FUNCTION_BLOCK CiA_DS402Statusword_INOVANCE EXTENDS CiA_DS402Statusword
VAR_INPUT
END_VAR
VAR_OUTPUT	
	TargetReached			: BOOL; // Bit 10 commonly used for in target position, velocity ect.
	HomeFound				: BOOL; // Bit 15: 
END_VAR

METHOD PUBLIC readStatusword : BOOL
VAR_INPUT
	Statusword 		:	UINT;
END_VAR
SUPER^.readStatusword(Statusword);

TargetReached												:= Statusword.10;
HomeFound													:= Statusword.15;
readStatusword												:= TRUE;
END_METHOD

END_FUNCTION_BLOCK

(* stored: Version 1.1.0.1, ProductVersion 3.1.4024.12
   POU CiA_DS402Statusword_INOVANCE: Id {050d2bb9-3b90-497f-8481-a04eace3b6fa}, SpecialFunc None
   Method readStatusword: Id {b2ce91d8-26fa-4160-9a5a-d3736baf5efb} *)
